// TwinCAT 3 PLC project plc_kfe_vac_vfs
// ProgramVersion: 3.1.4022.3
// libraries:
//   L2SI Vacuum Library, * (SLAC)
//   LCLS General, * (SLAC)
//   Tc2_Standard, * (Beckhoff Automation GmbH)
//   Tc2_System, * (Beckhoff Automation GmbH)
//   Tc3_Module, * (Beckhoff Automation GmbH)
//   PMPS,newest,SLAC - LCLS
// project tree:
//   GVLs/ GVL_SXR_VAC_Fast.TcGVL
//   / PlcTask.TcTTO
//   POUs/ MAIN.TcPOU, PRG_VFS.TcPOU

CONFIGURATION plc_kfe_vac_vfs
    RESOURCE PLC ON TwinCAT3
        TASK PlcTask(INTERVAL := T#150us, PRIORITY := 3);
        PROGRAM MAIN WITH PlcTask : MAIN;
    END_RESOURCE
END_CONFIGURATION

// ---- GVLs/GVL_SXR_VAC_Fast.TcGVL

VAR_GLOBAL
	
xSystemOverrideMode : BOOL; (* Global system override for the prototype section*)

fb_TV2K0_VFS_1 : FB_VFS;

END_VAR

// ---- POUs/MAIN.TcPOU
PROGRAM MAIN
VAR
	
	x: INT;
	y: INT;
	z: INT;
END_VAR

IF x > y THEN
	x := z;
ELSE
	x := x+1;
END_IF

PRG_VFS();

END_PROGRAM

// ---- POUs/PRG_VFS.TcPOU
PROGRAM PRG_VFS
VAR
END_VAR

fb_TV2K0_VFS_1(i_xOverrideMode := False, io_fbFFHWO =>);

END_PROGRAM
